{attribute 'qualified_only'}
VAR_GLOBAL CONSTANT
	// Mirrors Beckhoff's own Global_Version.stLibVersion_* pattern (see ST_LibVersion),
	// which only covers Tc2_*/Tc3_* library references, not custom ones -- until now: this
	// GVL uses Beckhoff's own naming exactly, so it merges into a consumer's Global_Version.
	// Kept in sync with <ProjectVersion> in HalfBROT.plcproj at release time.
	stLibVersion_HalfBROT : ST_LibVersion := (
		iMajor := 0,
		iMinor := 4,
		iBuild := 3,
		iRevision := 0,
		nFlags := 1,
		sVersion := '0.4.3'
	);
END_VAR

(* stored: Version 1.1.0.1, ProductVersion 3.1.4024.15
   GVL Global_Version: Id {6f45e4f1-e21a-4d69-b70c-b9b602163ca6} *)
